// TIA Portal V19 export
VAR_GLOBAL   // PLC tag table "2_BTRK_A0302_INGRESSO_CONST"
END_VAR
VAR_GLOBAL CONSTANT   // user constants
   BTRK_A0302_SPINTORE : Int := 1;   // Spintore ha iniziato la spinta verso la bordatrice
   BTRK_A0302_SPINTORE_USCITA_TRASPORTO_A031 : Int := 2;   // ... + il pezzo spinto ha raggiunto il sensore (xxxSQx) in uscita A03021
   BTRK_A0302_SPINTORE_INGRESSO_BORDATRICE : Int := 3;   // ... + Il pezzo è dentro la bordatrice ma non ha raggiunto ll secondo passaggio della bordatrice
   BTRK_A0302_INGRESSO_BORDATRICE : Int := 4;   // ... + Il pezzo è dentro la bordatrice e ha raggiunto ll secondo passaggio della bordatrice (spintore può ritornare indietro)
   BTRK_A0302_USCITA_BORDATRICE : Int := 5;   // il pezzo ha raggiunto il sensore di uscita della bordatrice (xxxSQx) (salvataggio posizione asse bordatrice)
   BTRK_A0302_USCITA_BORDATRICE_PAREG_CODA_BASSO : Int := 6;   // Il pezzo è in uscita della bordatrice ma la posizione target è limitata per non collidere con il pareggiamento di coda basso
   BTRK_A0302_USCITA_BORDATRICE_PAREG_CODA_ALTO : Int := 7;   // Il pezzo è in uscita della bordatrice e la posizione target non è limitata perchè il pareggiamento di coda è alto
END_VAR
